Fanuc KAREL source: kx00030.KL

-- PROVISIONAL review KL for V1013-1; original PC SHA256 efa09927ff236e5165f27b1f07b5dad4b8bad1f9e9b6488be13320eef024c5bd
-- Incomplete behavior may be omitted. Consult companion uncertainty JSON. Do not deploy.
PROGRAM KX00030
%NOLOCKGROUP
VAR
  I : INTEGER
  J : INTEGER
  B : BOOLEAN
  F : FILE
  S : STRING[80]
-- UNRESOLVED_DECL P type=000102
BEGIN
  -- UNRESOLVED_PC offsets 5-12; opcodes 9D,23
  -- UNRESOLVED_PC offsets 17-21; opcodes 7F
END KX00030
